(* IEC 61131-3 sources: volt/packages/volt-lsp-iec/test-corpus/awa-palletizer/Device/Plc Logic/Application/Library Manager/CmpIecVarAccess Implementation, 36 files *)

(* ---- SVN_INFO_FLAGS.gvl ---- *)
VAR_GLOBAL
	XINCOMPLETE : BOOL := FALSE;
	XMODIFIED : BOOL := TRUE;
	XSWITCHED : BOOL := FALSE;
	XCLEAN : BOOL := FALSE;
	XDISCONNECTED : BOOL := FALSE;
END_VAR

(* ---- SVN_INFO_LASTCHANGE.gvl ---- *)
VAR_GLOBAL
	DTLASTCHANGEUTC : DATE_AND_TIME := DATE_AND_TIME#2021-4-1-14:23:38;
	WSLASTCHANGELOCAL : WSTRING(44) := "2021-04-01 16:23:38 +0200 (Thu, 01 Apr 2021)";
	WSLASTCHANGEAUTHOR : WSTRING(8) := "b.schurr";
END_VAR

(* ---- SVN_INFO_REVISIONS.gvl ---- *)
VAR_GLOBAL
	LIMINREVISION : LINT := LINT#52494;
	LIMAXREVISION : LINT := LINT#52494;
END_VAR

(* ---- SVN_INFO_SUMMARY.gvl ---- *)
VAR_GLOBAL
	SVERSIONSUMMARY : STRING(6) := '52494M';
END_VAR

(* ---- SVN_INFO_SUMMARYW.gvl ---- *)
VAR_GLOBAL
	WSVERSIONSUMMARY : WSTRING(6) := "52494M";
END_VAR

(* ---- SVN_INFO_URI.gvl ---- *)
VAR_GLOBAL
	WURL : WSTRING(129) := "svn://server04/LibrariesV3Source/branches/V3.5.17.0/System/SysLibs/CmpIecVarAccess Implementation/CmpIecVarAccess Implementation/";
END_VAR

(* ---- IECVARACCBROWSEDOWN2.pou ---- *)
FUNCTION IECVARACCBROWSEDOWN2 : ICollections.IBaseTreeNode
VAR_INPUT
	HINTERFACE : SysTypes.RTS_IEC_HANDLE;
	HNODE : ICollections.IBaseTreeNode;
	PVARIABLEINFORMATION : POINTER TO IecVarAccess_Interfaces.VariableInformationStruct3;
	PRESULT : POINTER TO SysTypes.RTS_IEC_RESULT;
END_VAR
END_FUNCTION

(* ---- IECVARACCBROWSEGETNEXT2.pou ---- *)
FUNCTION IECVARACCBROWSEGETNEXT2 : ICollections.IBaseTreeNode
VAR_INPUT
	HINTERFACE : SysTypes.RTS_IEC_HANDLE;
	HNODE : ICollections.IBaseTreeNode;
	PVARIABLEINFORMATION : POINTER TO IecVarAccess_Interfaces.VariableInformationStruct3;
	PRESULT : POINTER TO SysTypes.RTS_IEC_RESULT;
END_VAR
END_FUNCTION

(* ---- IECVARACCBROWSERECURSIVE.pou ---- *)
FUNCTION IECVARACCBROWSERECURSIVE : SysTypes.RTS_IEC_RESULT
VAR_INPUT
	HINTERFACE : SysTypes.RTS_IEC_HANDLE;
	HNODE : ICollections.IBaseTreeNode;
	PVARIABLEINFORMATION : POINTER TO IecVarAccess_Interfaces.VariableInformationStruct3;
	PFBROWSECALLBACK : POINTER TO BYTE;
	PUSERPARAMETER : POINTER TO BYTE;
END_VAR
END_FUNCTION

(* ---- IECVARACCBROWSEUP2.pou ---- *)
FUNCTION IECVARACCBROWSEUP2 : ICollections.IBaseTreeNode
VAR_INPUT
	HINTERFACE : SysTypes.RTS_IEC_HANDLE;
	HNODE : ICollections.IBaseTreeNode;
	PVARIABLEINFORMATION : POINTER TO IecVarAccess_Interfaces.VariableInformationStruct3;
	PRESULT : POINTER TO SysTypes.RTS_IEC_RESULT;
END_VAR
END_FUNCTION

(* ---- IECVARACCEXITVARINFO.pou ---- *)
FUNCTION IECVARACCEXITVARINFO : SysTypes.RTS_IEC_RESULT
VAR_INPUT
	PVARIABLEINFORMATION : POINTER TO IecVarAccess_Interfaces.VariableInformationStruct3;
END_VAR
END_FUNCTION

(* ---- IECVARACCGETFIRSTINTERFACE.pou ---- *)
FUNCTION IECVARACCGETFIRSTINTERFACE : IIecVarAccess3
VAR_INPUT
	PRESULT : POINTER TO RTS_IEC_RESULT;
END_VAR
END_FUNCTION

(* ---- IECVARACCGETFIRSTINTERFACE2.pou ---- *)
FUNCTION IECVARACCGETFIRSTINTERFACE2 : IBase
VAR_INPUT
	PRESULT : POINTER TO RTS_IEC_RESULT;
END_VAR
END_FUNCTION

(* ---- IECVARACCGETNEXTINTERFACE.pou ---- *)
FUNCTION IECVARACCGETNEXTINTERFACE : IIecVarAccess3
VAR_INPUT
	PIPREV : IIecVarAccess3;
	PRESULT : POINTER TO RTS_IEC_RESULT;
END_VAR
END_FUNCTION

(* ---- IECVARACCGETNEXTINTERFACE2.pou ---- *)
FUNCTION IECVARACCGETNEXTINTERFACE2 : IBase
VAR_INPUT
	PIPREV : IBase;
	PRESULT : POINTER TO RTS_IEC_RESULT;
END_VAR
END_FUNCTION

(* ---- IECVARACCGETNODE4.pou ---- *)
FUNCTION IECVARACCGETNODE4 : ICollections.IBaseTreeNode
VAR_INPUT
	PSZPATH : POINTER TO STRING;
	PHINTERFACE : POINTER TO SysTypes.RTS_IEC_HANDLE;
	PVARIABLEINFORMATION : POINTER TO IecVarAccess_Interfaces.VariableInformationStruct3;
	PRESULT : POINTER TO SysTypes.RTS_IEC_RESULT;
END_VAR
END_FUNCTION

(* ---- IECVARACCGETNODEFULLPATH4.pou ---- *)
FUNCTION IECVARACCGETNODEFULLPATH4 : DINT
VAR_INPUT
	HINTERFACE : SysTypes.RTS_IEC_HANDLE;
	HNODE : ICollections.IBaseTreeNode;
	PVARIABLEINFORMATION : POINTER TO IecVarAccess_Interfaces.VariableInformationStruct3;
	PSZPATH : POINTER TO STRING;
	IMAXPATH : DINT;
	PRESULT : POINTER TO SysTypes.RTS_IEC_RESULT;
END_VAR
END_FUNCTION

(* ---- IECVARACCGETNODENAME4.pou ---- *)
FUNCTION IECVARACCGETNODENAME4 : SysTypes.RTS_IEC_RESULT
VAR_INPUT
	HINTERFACE : SysTypes.RTS_IEC_HANDLE;
	HNODE : ICollections.IBaseTreeNode;
	PVARIABLEINFORMATION : POINTER TO IecVarAccess_Interfaces.VariableInformationStruct3;
	PSZNODENAME : POINTER TO STRING;
	NNODENAMELEN : UDINT;
END_VAR
END_FUNCTION

(* ---- IECVARACCGETSYMBOLSETMASK.pou ---- *)
FUNCTION IECVARACCGETSYMBOLSETMASK : DWORD
VAR_INPUT
	HUSER : RTS_IEC_HANDLE;
	HINTERFACE : RTS_IEC_HANDLE;
	PRESULT : POINTER TO RTS_IEC_RESULT;
END_VAR
END_FUNCTION

(* ---- IECVARACCINITVARINFO.pou ---- *)
FUNCTION IECVARACCINITVARINFO : SysTypes.RTS_IEC_RESULT
VAR_INPUT
	PVARIABLEINFORMATION : POINTER TO IecVarAccess_Interfaces.VariableInformationStruct3;
	NSIZEOFVARINFO : UINT;
END_VAR
END_FUNCTION

(* ---- IECVARACCINITVARINFO2.pou ---- *)
FUNCTION IECVARACCINITVARINFO2 : SysTypes.RTS_IEC_RESULT
VAR_INPUT
	PVARIABLEINFORMATION : POINTER TO IecVarAccess_Interfaces.VariableInformationStruct3;
	NSIZEOFVARINFO : UINT;
	HUSER : RTS_IEC_HANDLE;
END_VAR
END_FUNCTION

(* ---- IECVARACCINVALIDATENODE.pou ---- *)
FUNCTION IECVARACCINVALIDATENODE : RTS_IEC_RESULT
VAR_INPUT
	HNODE : RTS_IEC_HANDLE;
END_VAR
END_FUNCTION

(* ---- IECVARACCNODEINFOADDBROWSEINFO.pou ---- *)
FUNCTION IECVARACCNODEINFOADDBROWSEINFO : SysTypes.RTS_IEC_RESULT
VAR_INPUT
	PVARIABLEINFORMATION : POINTER TO IecVarAccess_Interfaces.VariableInformationStruct3;
	PBROWSEINFODATA : POINTER TO RtsBrowseInfo;
END_VAR
END_FUNCTION

(* ---- IECVARACCNODEINFOADDREFERENCE.pou ---- *)
FUNCTION IECVARACCNODEINFOADDREFERENCE : SysTypes.RTS_IEC_RESULT
VAR_INPUT
	PVARIABLEINFORMATION : POINTER TO IecVarAccess_Interfaces.VariableInformationStruct3;
	PREFERENCEINFODATA : POINTER TO BYTE;
	NINFOSIZE : XWORD;
	PNEWREFERENCEINFO : POINTER TO POINTER TO BYTE;
END_VAR
END_FUNCTION

(* ---- IECVARACCNODEINFOGETBROWSEINFO.pou ---- *)
FUNCTION IECVARACCNODEINFOGETBROWSEINFO : POINTER TO RtsBrowseInfo
VAR_INPUT
	PVARIABLEINFORMATION : POINTER TO IecVarAccess_Interfaces.VariableInformationStruct3;
	PLAST : POINTER TO RtsBrowseInfo;
	PRESULT : POINTER TO SysTypes.RTS_IEC_RESULT;
END_VAR
END_FUNCTION

(* ---- IECVARACCNODEINFOGETREFERENCE.pou ---- *)
FUNCTION IECVARACCNODEINFOGETREFERENCE : POINTER TO BYTE
VAR_INPUT
	PVARIABLEINFORMATION : POINTER TO IecVarAccess_Interfaces.VariableInformationStruct3;
	PRESULT : POINTER TO SysTypes.RTS_IEC_RESULT;
END_VAR
END_FUNCTION

(* ---- IECVARACCNODEINFOREMOVEBROWSEINFO.pou ---- *)
FUNCTION IECVARACCNODEINFOREMOVEBROWSEINFO : SysTypes.RTS_IEC_RESULT
VAR_INPUT
	PVARIABLEINFORMATION : POINTER TO IecVarAccess_Interfaces.VariableInformationStruct3;
END_VAR
END_FUNCTION

(* ---- IECVARACCNODEINFOREMOVEREFERENCE.pou ---- *)
FUNCTION IECVARACCNODEINFOREMOVEREFERENCE : SysTypes.RTS_IEC_RESULT
VAR_INPUT
	PVARIABLEINFORMATION : POINTER TO IecVarAccess_Interfaces.VariableInformationStruct3;
END_VAR
END_FUNCTION

(* ---- IECVARACCREGISTERINSTANCE.pou ---- *)
FUNCTION IECVARACCREGISTERINSTANCE : RTS_IEC_HANDLE
VAR_INPUT
	PIIECVARACCESS : CmpIecVarAccess_Interfaces.IIecVarAccess;
	PRESULT : POINTER TO RTS_IEC_RESULT;
END_VAR
END_FUNCTION

(* ---- IECVARACCREGISTERINSTANCE2.pou ---- *)
FUNCTION IECVARACCREGISTERINSTANCE2 : RTS_IEC_HANDLE
VAR_INPUT
	PIIECVARACCESS2 : CmpIecVarAccess_Interfaces.IIecVarAccess2;
	PRESULT : POINTER TO RTS_IEC_RESULT;
END_VAR
END_FUNCTION

(* ---- IECVARACCREGISTERINSTANCE3.pou ---- *)
FUNCTION IECVARACCREGISTERINSTANCE3 : RTS_IEC_HANDLE
VAR_INPUT
	PIIECVARACCESS3 : IIecVarAccess3;
	PRESULT : POINTER TO RTS_IEC_RESULT;
END_VAR
END_FUNCTION

(* ---- IECVARACCREGISTERINSTANCEBASE.pou ---- *)
FUNCTION IECVARACCREGISTERINSTANCEBASE : RTS_IEC_HANDLE
VAR_INPUT
	PIBASE : IBase;
	PRESULT : POINTER TO RTS_IEC_RESULT;
END_VAR
END_FUNCTION

(* ---- IECVARACCREGISTERINSTANCEBASE2.pou ---- *)
FUNCTION IECVARACCREGISTERINSTANCEBASE2 : RTS_IEC_HANDLE
VAR_INPUT
	PIBASE : IBase;
	UDICRC : UDINT;
	PRESULT : POINTER TO RTS_IEC_RESULT;
END_VAR
END_FUNCTION

(* ---- IECVARACCSETSYMBOLCONFIGCRC.pou ---- *)
FUNCTION IECVARACCSETSYMBOLCONFIGCRC : RTS_IEC_RESULT
VAR_INPUT
	HINSTANCE : RTS_IEC_HANDLE;
	UDICRC : UDINT;
END_VAR
END_FUNCTION

(* ---- IECVARACCUNREGISTERINSTANCE.pou ---- *)
FUNCTION IECVARACCUNREGISTERINSTANCE : RTS_IEC_RESULT
VAR_INPUT
	HINSTANCE : RTS_IEC_HANDLE;
END_VAR
END_FUNCTION

(* ---- IECVARACCUPDATESYMBOLSETS.pou ---- *)
FUNCTION IECVARACCUPDATESYMBOLSETS : RTS_IEC_RESULT
VAR_INPUT
	HINTERFACE : RTS_IEC_HANDLE;
	PSYMBOLSSETS : POINTER TO IecVarAccSymbolSetDescription;
	NUMOFSYMBOLSSETS : UDINT;
END_VAR
END_FUNCTION
